TYPE ST_TsFbInfo :
STRUCT
	
	nState  								:USINT;
	nDiag  									:UINT;

END_STRUCT
END_TYPE
(* End *)

(* stored: Version 1.1.0.1, ProductVersion 3.1.4022.16
   DUT ST_TsFbInfo: Id {566c886e-fc70-4dd7-9ca6-2fb5c62046fe} *)
